Fanuc KAREL source: kf00106.KL

-- PROVISIONAL review KL for V940-1; original PC SHA256 22cca7ff2c6838cd8d2269c20ee17609596ed0e899e908e95609621312b90f2f
-- Incomplete behavior may be omitted. Consult companion uncertainty JSON. Do not deploy.
PROGRAM KF00106
%NOLOCKGROUP
BEGIN
  -- V9_ZERO_TABLE_METADATA_HINT layout=0002_ascii; no indexed target words; source/name/runtime held
  -- UNRESOLVED_PC offsets 5-16; opcodes 2E,23
  -- UNRESOLVED_PC offsets 21-32; opcodes 2E,23
  -- UNRESOLVED_PC offsets 37-57; opcodes 27,27,9D,22,2A,22,31
  -- UNRESOLVED_PC offsets 62-66; opcodes 7F
END KF00106
